// TwinCAT 3 PLC project PLC
// ProgramVersion: 3.1.4026.20
// CompilerDefines: VISU_USEPROPERTYINFO
// libraries:
//   SPT Base Types, * (Beckhoff Automation LLC)
//   SPT Components, * (Beckhoff Automation LLC)
//   SPT Diagnostic, * (Beckhoff Automation LLC)
//   SPT EtherCat, * (Beckhoff Automation LLC)
//   SPT Event Logger, * (Beckhoff Automation LLC)
//   SPT Motion Control, * (Beckhoff Automation LLC)
//   SPT Utilities, * (Beckhoff Automation LLC)
//   Tc2_MC2, * (Beckhoff Automation GmbH)
//   Tc2_MC2_Camming, * (Beckhoff Automation GmbH)
//   Tc2_Standard, * (Beckhoff Automation GmbH)
//   Tc2_System, * (Beckhoff Automation GmbH)
//   Tc2_Utilities, * (Beckhoff Automation GmbH)
//   Tc3_EventLogger, * (Beckhoff Automation GmbH)
//   Tc3_MC2_AdvancedHoming, * (Beckhoff Automation GmbH)
//   Tc3_McCollisionAvoidance, * (Beckhoff Automation GmbH)
//   Tc3_McCoordinatedMotion, * (Beckhoff Automation GmbH)
//   Tc3_PackML_V3, * (Beckhoff Automation GmbH)
// project tree:
//   / GlobalTextList.TcGTLO, PlcTask.TcTTO (not stored), VisualizationManager.TcVMO (not stored)
//   GVLs/ GVL.TcGVL (not stored)
//   POUs/BeltIndexer/ FB_DataSetFifo.TcPOU (not stored), FB_BeltIndexer.TcPOU
//   POUs/Camming/02 Cam Module Update Table/ CamModule_UpdateTable.TcPOU (not stored)
//   POUs/Camming/02 Cam Module Update Table/DUTs/ ST_EM_Cfg_UpdateTable.TcDUT, ST_EM_Cmd_UpdateTable.TcDUT, ST_EM_HMI_UpdateTable.TcDUT (not stored), ST_EM_Sts_UpdateTable.TcDUT
//   POUs/ Machine.TcPOU (not stored), MAIN.TcPOU (not stored)
//   POUs/RackAndPinion/ FB_RackAndPinion.TcPOU, FB_SwitchHoming.TcPOU, FB_TorqueHoming.TcPOU
//   POUs/Stitcher/ FB_Stitcher.TcPOU (not stored)
//   VISUs/ Visualization.TcVIS (not stored)

// ---- POUs/Camming/02 Cam Module Update Table/DUTs/ST_EM_Cfg_UpdateTable.TcDUT
TYPE ST_EM_Cfg_UpdateTable :
	STRUCT
		CamActivationMode : INT;
	END_STRUCT
END_TYPE

// ---- POUs/Camming/02 Cam Module Update Table/DUTs/ST_EM_Cmd_UpdateTable.TcDUT
TYPE ST_EM_Cmd_UpdateTable :
	STRUCT
		ChangeTable : BOOL;
		ChangeMode	: BOOL;
	END_STRUCT
END_TYPE

// ---- POUs/Camming/02 Cam Module Update Table/DUTs/ST_EM_Sts_UpdateTable.TcDUT
TYPE ST_EM_Sts_UpdateTable :
	STRUCT
		CurrentTable : UDINT;
	END_STRUCT
END_TYPE

// ---- POUs/RackAndPinion/FB_RackAndPinion.TcPOU
FUNCTION_BLOCK FB_RackAndPinion EXTENDS FB_PackML_BaseModule
VAR
	LeftAxis	: FB_Component_BasicAxis;
	RightAxis	: FB_Component_BasicAxis;

	TorqueHoming	: FB_TorqueHoming;
	SwitchHoming	: FB_SwitchHoming;

	// CA Group
	CAGroup			: AXES_GROUP_REF;
	GroupReadStatus	: MC_GroupReadStatus;
	GroupReset		: MC_GroupReset;
	GroupEnable		: MC_GroupEnable;
	GroupDisable	: MC_GroupDisable;
	AddToGroup		: ARRAY[0..1] OF MC_AddAxisToGroup;
	MoveAbsoluteCA	: ARRAY[0..1] OF MC_MoveAbsoluteCA;

	TON_Dwell	: TON;
END_VAR

//! @summary This method contains code which will execute when this PackML module is in the <b>Aborting</b> state
METHOD PROTECTED Aborting
VAR
	i				: UDINT;
	SubModulesReady : BOOL := TRUE;
END_VAR
CASE DescendantSequenceState OF
	0:
		NoStateTasksToComplete := FALSE;
		DescendantSequenceState := DescendantSequenceState + 10;

	10:
		IF LeftAxis.Disable() AND RightAxis.Disable() THEN
			StateTasksComplete 		:= TRUE;
			DescendantSequenceState := DescendantSequenceState + 10;
		END_IF

	//20:	

	20:
		StateTasksComplete := TRUE;
END_CASE

SUPER^.Aborting();
END_METHOD

//! @summary This method contains code which will execute when this PackML module is in the <b>Clearing</b> state
METHOD PROTECTED Clearing
VAR
	i				: UDINT;
	SubModulesReady : BOOL := TRUE;
END_VAR

VAR_INST

END_VAR

(*! <description> <b>Note:</b> The <i>Clear</i> command can also be thought of as a <i>fault reset</i> depite the ambiguity in the naming of the <i>Reset</i> state. 
<table> 
	<tr>
		<th> Previous State </th>
		<th> Transition In </th>
		<th> Transition Out </th>
		<th> Next State  </th> 
	</tr>
	<tr>
		<td> Aborted </td>
		<td> Clear Command </td> 
		<td> State Complete </td>
		<td> Stopped </td> 
	</tr>
</table>
This method is called as required by <c>StateControl()</c>
</description> 

*)
// CASE _CurrentMode OF
// 	E_PMLUnitMode.ePMLUnitMode_Production:
		CASE DescendantSequenceState OF
			0: //Init
				NoStateTasksToComplete := FALSE;

				//Reset Axes and  CA Group
				LeftAxis.Reset();
				RightAxis.Reset();
				GroupReset.Execute	:= TRUE;
				DescendantSequenceState := DescendantSequenceState + 10;

			10: // Done	
				GroupReset.Execute	:= FALSE;
				StateTasksComplete := TRUE;
		END_CASE

// END_CASE

SUPER^.Clearing();
END_METHOD

METHOD CyclicLogic
VAR_INPUT
END_VAR
SUPER^.CyclicLogic();

AddToGroup[0](Axis := LeftAxis.Axis, AxesGroup := CAGroup);
AddToGroup[1](Axis := RightAxis.Axis, AxesGroup := CAGroup);
GroupEnable(AxesGroup := CAGroup);
GroupDisable(AxesGroup := CAGroup);
GroupReadStatus.Enable		:= TRUE;
GroupReadStatus(AxesGroup	:= CAGroup);
GroupReset(AxesGroup	:= CAGroup);
MoveAbsoluteCA[0](Axis := LeftAxis.Axis);
MoveAbsoluteCA[1](Axis := RightAxis.Axis);
TON_Dwell();

TorqueHoming.CyclicLogic();
SwitchHoming.CyclicLogic();
END_METHOD

//! @summary This method contains code which will execute when this PackML module is in the <b>Execute</b> state
METHOD PROTECTED Execute
VAR
	i : UDINT;
END_VAR
(*CASE _CurrentMode OF
	E_PMLUnitMode.ePMLUnitMode_Production:


	E_PMLUnitMode.ePMLUnitMode_Manual:
		; //Insert logic for Manual Mode here
END_CASE	*)

CASE DescendantSequenceState OF
	0:
		FOR i := 0 TO 1 DO
			MoveAbsoluteCA[i].Execute		:= TRUE;
			MoveAbsoluteCA[i].Position		:= 50.0;
			MoveAbsoluteCA[i].Velocity		:= leftAxis.Velocity;
			MoveAbsoluteCA[i].Acceleration	:= LeftAxis.Acceleration;
			MoveAbsoluteCA[i].Deceleration	:= LeftAxis.Deceleration;
			MoveAbsoluteCA[i].Jerk			:= LeftAxis.Jerk;
			MoveAbsoluteCA[i].Gap			:= 68.0;
			MoveAbsoluteCA[i].Options.GapControlMode	:= MC_GAP_CONTROL_MODE.mcGapControlModeFast;
			MoveAbsoluteCA[i].BufferMode	:= mcAborting;
		END_FOR
		DescendantSequenceState				:= DescendantSequenceState + 10;

	10:	IF MoveAbsoluteCA[0].Done OR MoveAbsoluteCA[1].Done THEN
			MoveAbsoluteCA[0].Execute		:= FALSE;
			MoveAbsoluteCA[1].Execute		:= FALSE;
			TON_Dwell.IN	:= TRUE;
			TON_Dwell.PT	:= T#1S;
			DescendantSequenceState			:= DescendantSequenceState + 10;
		END_IF

	20: IF TON_Dwell.Q THEN
			ton_dwell.IN	:= FALSE;
			DescendantSequenceState			:= DescendantSequenceState + 10;
		END_IF

	30:
		FOR i := 0 TO 1 DO
			MoveAbsoluteCA[i].Execute		:= TRUE;
			MoveAbsoluteCA[i].Position		:= 450.0;
			MoveAbsoluteCA[i].Velocity		:= leftAxis.Velocity;
			MoveAbsoluteCA[i].Acceleration	:= LeftAxis.Acceleration;
			MoveAbsoluteCA[i].Deceleration	:= LeftAxis.Deceleration;
			MoveAbsoluteCA[i].Jerk			:= LeftAxis.Jerk;
			MoveAbsoluteCA[i].Gap			:= 68.0;
			MoveAbsoluteCA[i].Options.GapControlMode	:= MC_GAP_CONTROL_MODE.mcGapControlModeStandard;
			MoveAbsoluteCA[i].BufferMode	:= mcAborting;
		END_FOR
		DescendantSequenceState				:= DescendantSequenceState + 10;

	40:	IF MoveAbsoluteCA[0].Done OR MoveAbsoluteCA[1].Done THEN
			MoveAbsoluteCA[0].Execute		:= FALSE;
			MoveAbsoluteCA[1].Execute		:= FALSE;
			TON_Dwell.IN	:= TRUE;
			TON_Dwell.PT	:= T#1S;
			DescendantSequenceState			:= DescendantSequenceState + 10;

		END_IF

	50: IF TON_Dwell.Q THEN
			ton_dwell.IN	:= FALSE;
			DescendantSequenceState			:= 0;
		END_IF

END_CASE
END_METHOD

(* Basic module initialization logic*)
METHOD PROTECTED Initialize : BOOL
Initialize := FALSE;
CASE DescendantSequenceState OF
	0:
		RegisterComponent(Component := LeftAxis);
		RegisterComponent(Component := RightAxis);
		DescendantSequenceState := DescendantSequenceState + 10;

	10:
		IF SUPER^.Initialize() THEN
			DescendantSequenceState := DescendantSequenceState + 10;
		END_IF

	20:
		Initialize := TRUE;
END_CASE
END_METHOD

METHOD PROTECTED Resetting
VAR_INST
	i			 : UDINT;
END_VAR
// CASE _CurrentMode OF
// 	E_PMLUnitMode.ePMLUnitMode_Production:
		CASE DescendantSequenceState OF
			0: //Init
				i					   := 1;
				NoStateTasksToComplete := FALSE;
				DescendantSequenceState := DescendantSequenceState + 10;

			10: //Enable Axes
				IF LeftAxis.Enable() AND RightAxis.Enable() THEN
					DescendantSequenceState := DescendantSequenceState + 10;
				END_IF

			// Add logic to home left axis to switch and right axis to hard stop
			20: // Home Right Axis
				TorqueHoming.Axis	:= RightAxis;
				SwitchHoming.Axis	:= LeftAxis;
				IF TorqueHoming.Execute() AND SwitchHoming.Execute() THEN
					DescendantSequenceState := DescendantSequenceState + 20;
				END_IF

			30:	// Home Left Axis
				SwitchHoming.Axis	:= LeftAxis;
				IF SwitchHoming.Execute() THEN
					DescendantSequenceState := DescendantSequenceState + 10;
				END_IF

			40: //Add Movers to Group			
				AddToGroup[0].Execute		:= AddToGroup[1].Execute		:= TRUE;
				AddToGroup[0].IdentInGroup	:= UDINT_TO_IDENTINGROUP(1);
				AddToGroup[1].IdentInGroup	:= UDINT_TO_IDENTINGROUP(2);
				IF AddToGroup[0].Done AND AddToGroup[1].Done THEN	
					AddToGroup[0].Execute	:= AddToGroup[1].Execute	:= FALSE;
					DescendantSequenceState := DescendantSequenceState + 10;
				END_IF

			50: //Enable CA Group
				GroupEnable.Execute	:= TRUE;
				IF GroupEnable.Done THEN
					DescendantSequenceState := DescendantSequenceState + 10;
				END_IF

			60: //Clearing complete
				StateTasksComplete := TRUE;

		END_CASE
// END_CASE

SUPER^.Resetting();
END_METHOD

METHOD PROTECTED Starting
VAR_INST
	i		  : UDINT;
END_VAR
//CASE _CurrentMode OF
//	E_PMLUnitMode.ePMLUnitMode_Production:
		CASE DescendantSequenceState OF
			0:
				NoStateTasksToComplete	:= FALSE;
				DescendantSequenceState := 10;
				i						:= 1;

			10: //Set Axis Parameters
				LeftAxis.Velocity		:= 250;		RightAxis.Velocity		:= 250;
				LeftAxis.Acceleration	:= 1000;	RightAxis.Acceleration	:= 1000;
				LeftAxis.Deceleration	:= 1000;	RightAxis.Deceleration	:= 1000;
				LeftAxis.Jerk			:= 10000;	RightAxis.Jerk			:= 10000;
				DescendantSequenceState := DescendantSequenceState + 10;
				StateTasksComplete 		:= TRUE;

			20: //Cleanup mover queues
				DescendantSequenceState := DescendantSequenceState + 10;

		END_CASE

	//E_PMLUnitMode.ePMLUnitMode_Manual:
//END_CASE

SUPER^.Starting();
END_METHOD

END_FUNCTION_BLOCK

// ---- POUs/RackAndPinion/FB_TorqueHoming.TcPOU
FUNCTION_BLOCK FB_TorqueHoming IMPLEMENTS I_MotionSequence
VAR_INPUT
	HomingParameter	: MC_HomingParameter;
END_VAR
VAR_OUTPUT
	State	: UINT;
END_VAR
VAR
	validaxisref	: BOOL := FALSE;
	_Axis			: SPT_Motion_Control.I_BasicAxis;
	StepBlockHoming	: MC_StepBlock;
	FinishHoming	: MC_FinishHoming;
END_VAR

{warning 'Add property implementation'}
PROPERTY Axis : SPT_Motion_Control.I_BasicAxis
GET
Axis	:= _Axis;
END_GET
SET
_Axis	:= Axis;
validaxisref	:= TRUE;
END_SET
END_PROPERTY

{warning 'Add property implementation'}
PROPERTY Busy : BOOL
GET
END_GET
END_PROPERTY

{warning 'Add method implementation '}
METHOD CyclicLogic
IF validaxisref THEN
	StepBlockHoming(Axis := _Axis.Axis, Parameter := HomingParameter);
	FinishHoming(Axis := _Axis.Axis, Parameter := HomingParameter);
END_IF

IF NOT StepBlockHoming.Execute	THEN
	State	:= 0;
END_IF
StepBlockHoming.Execute	:= FALSE;
FinishHoming.Execute	:= FALSE;
END_METHOD

{warning 'Add property implementation'}
PROPERTY Error : BOOL
GET
END_GET
END_PROPERTY

{warning 'Add property implementation'}
PROPERTY ErrorID : UDINT
GET
END_GET
END_PROPERTY

{warning 'Add method implementation '}
METHOD Execute : BOOL
StepBlockHoming.Execute					:= TRUE;
StepBlockHoming.SetPosition				:= 472;
StepBlockHoming.Direction				:= mcPositiveDirection;
StepBlockHoming.Velocity				:= 50;
StepBlockHoming.Acceleration			:= 1000;
StepBlockHoming.Deceleration			:= 1000;
StepBlockHoming.Jerk					:= 10000;
StepBlockHoming.DetectionVelocityLimit	:= 1;
StepBlockHoming.DetectionVelocityTime	:= T#100MS;
StepBlockHoming.TimeLimit				:= T#10S;
StepBlockHoming.DistanceLimit			:= 500;
StepBlockHoming.TorqueLimit				:= 50;
StepBlockHoming.TorqueTolerance			:= 5;

FinishHoming.Execute		:= StepBlockHoming.Done;
FinishHoming.Distance		:= -0.5;
FinishHoming.Velocity		:= 100;
FinishHoming.Acceleration	:= 1000;
FinishHoming.Deceleration	:= 1000;
FinishHoming.Jerk			:= 1000;

// return true when done
Execute	:= StepBlockHoming.Done AND FinishHoming.Done;
END_METHOD

{warning 'Add property implementation'}
PROPERTY InitComplete : BOOL
GET
END_GET
END_PROPERTY

END_FUNCTION_BLOCK

// ---- POUs/RackAndPinion/FB_SwitchHoming.TcPOU
FUNCTION_BLOCK FB_SwitchHoming IMPLEMENTS I_MotionSequence
VAR_INPUT
	HomingParameter	: MC_HomingParameter;
END_VAR
VAR_OUTPUT
	State	: UINT;
END_VAR
VAR
	diHomeSwitch	AT %I* : BOOL;
	doHomeSwitch	AT %Q* : BOOL := TRUE;
	validaxisref	: BOOL := FALSE;
	_Axis			: SPT_Motion_Control.I_BasicAxis;
	Home			: MC_Home;
END_VAR

{warning 'Add property implementation'}
PROPERTY Axis : SPT_Motion_Control.I_BasicAxis
GET
Axis	:= _Axis;
END_GET
SET
_Axis	:= Axis;
validaxisref	:= TRUE;
END_SET
END_PROPERTY

{warning 'Add property implementation'}
PROPERTY Busy : BOOL
GET
END_GET
END_PROPERTY

{warning 'Add method implementation '}
METHOD CyclicLogic
IF validaxisref THEN
	Home.bCalibrationCam	:= diHomeSwitch;
	Home(Axis := _Axis.Axis);

END_IF

IF NOT Home.Execute	THEN
	State	:= 0;
END_IF
Home.Execute	:= FALSE;
END_METHOD

{warning 'Add property implementation'}
PROPERTY Error : BOOL
GET
END_GET
END_PROPERTY

{warning 'Add property implementation'}
PROPERTY ErrorID : UDINT
GET
END_GET
END_PROPERTY

{warning 'Add method implementation '}
METHOD Execute : BOOL
Home.Execute					:= TRUE;
Home.Position					:= 39;
Home.HomingMode					:= MC_DefaultHoming;
Home.Options.SearchVelocity		:= 50;
Home.Options.SearchDirection	:= MC_Negative_Direction;

// return true when done
Execute	:= Home.Done;
END_METHOD

{warning 'Add property implementation'}
PROPERTY InitComplete : BOOL
GET
END_GET
END_PROPERTY

END_FUNCTION_BLOCK

// ---- POUs/BeltIndexer/FB_BeltIndexer.TcPOU
FUNCTION_BLOCK FB_BeltIndexer EXTENDS FB_PackML_BaseModule
VAR
	BeltAxis	: FB_Component_BasicAxis;

	TouchProbe			: MC_TouchProbe;
	TouchProbeConfig	: TRIGGER_REF;
	fbFifo 				: FB_DataSetFifo := ( bOverwrite := TRUE );
	arrBuffer 			: ARRAY[0..MAX_BUFFER_SIZE] OF BYTE; (* Buffer memory used by FB_MemRingBuffer function block *)

	NewRecordedPosition	: LREAL;
	OldRecordedPosition	: LREAL;

	TON_Dwell	: TON;
END_VAR

//! @summary This method contains code which will execute when this PackML module is in the <b>Aborting</b> state
METHOD PROTECTED Aborting
VAR
	i				: UDINT;
	SubModulesReady : BOOL := TRUE;
END_VAR
CASE DescendantSequenceState OF
	0:
		NoStateTasksToComplete := FALSE;
		DescendantSequenceState := DescendantSequenceState + 10;

	10:
		IF BeltAxis.Disable() THEN
			TouchProbe.Execute		:= FALSE;
			NewRecordedPosition		:= 0;
			OldRecordedPosition		:= 0;
			StateTasksComplete 		:= TRUE;
			DescendantSequenceState := DescendantSequenceState + 10;
		END_IF

	//20:	

	20:
		StateTasksComplete := TRUE;
END_CASE

SUPER^.Aborting();
END_METHOD

//! @summary This method contains code which will execute when this PackML module is in the <b>Clearing</b> state
METHOD PROTECTED Clearing
VAR
	i				: UDINT;
	SubModulesReady : BOOL := TRUE;
END_VAR

VAR_INST

END_VAR

(*! <description> <b>Note:</b> The <i>Clear</i> command can also be thought of as a <i>fault reset</i> depite the ambiguity in the naming of the <i>Reset</i> state. 
<table> 
	<tr>
		<th> Previous State </th>
		<th> Transition In </th>
		<th> Transition Out </th>
		<th> Next State  </th> 
	</tr>
	<tr>
		<td> Aborted </td>
		<td> Clear Command </td> 
		<td> State Complete </td>
		<td> Stopped </td> 
	</tr>
</table>
This method is called as required by <c>StateControl()</c>
</description> 

*)
// CASE _CurrentMode OF
// 	E_PMLUnitMode.ePMLUnitMode_Production:
		CASE DescendantSequenceState OF
			0: //Init
				NoStateTasksToComplete := FALSE;

				//Reset Axes and  CA Group
				BeltAxis.Reset();
				DescendantSequenceState := DescendantSequenceState + 10;

			10: // Done	
				StateTasksComplete := TRUE;
		END_CASE

// END_CASE

SUPER^.Clearing();
END_METHOD

METHOD CyclicLogic
VAR_INPUT
END_VAR
SUPER^.CyclicLogic();

TouchProbe(Axis := BeltAxis.Axis, TriggerInput := TouchProbeConfig);
fbFifo();
TON_Dwell();
END_METHOD

//! @summary This method contains code which will execute when this PackML module is in the <b>Execute</b> state
METHOD PROTECTED Execute
VAR
	i : UDINT;
END_VAR
(*CASE _CurrentMode OF
	E_PMLUnitMode.ePMLUnitMode_Production:


	E_PMLUnitMode.ePMLUnitMode_Manual:
		; //Insert logic for Manual Mode here
END_CASE	*)

CASE DescendantSequenceState OF
	0:	// Start Moving
		BeltAxis.MoveVelocity(250, TRUE);
		TouchProbe.Execute		:= TRUE;
		DescendantSequenceState	:= DescendantSequenceState + 10;

	10: // Start buffering positions and moving to them
		IF fbFifo.nCount > 0 THEN
			fbFifo.A_Get(out => OldRecordedPosition);
			BeltAxis.MoveAbsolute(OldRecordedPosition + 440.0, TRUE);
			DescendantSequenceState	:= DescendantSequenceState + 10;
		END_IF
		
	20: // Look for trigger
		IF ton_dwell.Q THEN
			TON_Dwell.IN			:= FALSE;
			fbFifo.A_Remove();
			IF fbFifo.nCount > 0 THEN
				DescendantSequenceState	:= 10;
			ELSE
				DescendantSequenceState	:= 0;
			END_IF
		ELSIF BeltAxis.InPosition AND (ABS(BeltAxis.SetPosition - (OldRecordedPosition + 440)) < 1) THEN
			Ton_Dwell.IN	:= TRUE;
		END_IF

END_CASE

IF TouchProbe.Done THEN
	NewRecordedPosition	:= TouchProbe.RecordedData.AbsolutePosition;
	fbFifo.A_Add(In := NewRecordedPosition);
END_IF
END_METHOD

(* Basic module initialization logic*)
METHOD PROTECTED Initialize : BOOL
Initialize := FALSE;
CASE DescendantSequenceState OF
	0:
		RegisterComponent(Component := BeltAxis);
		DescendantSequenceState := DescendantSequenceState + 10;

	10: // Touch Probe Configuration
		TouchProbeConfig.SignalSource	:= SignalSource_DriveDefined;
		TouchProbeconfig.Mode			:= TOUCHPROBEMODE_CONTINOUS;
		TON_Dwell.PT					:= T#500ms;
		DescendantSequenceState 		:= DescendantSequenceState + 10;

	20:
		IF SUPER^.Initialize() THEN
			DescendantSequenceState := DescendantSequenceState + 10;
		END_IF

	30:
		Initialize := TRUE;
END_CASE
END_METHOD

METHOD PROTECTED Resetting
VAR_INST
	i			 : UDINT;
END_VAR
// CASE _CurrentMode OF
// 	E_PMLUnitMode.ePMLUnitMode_Production:
		CASE DescendantSequenceState OF
			0: //Init
				i					   := 1;
				NoStateTasksToComplete := FALSE;
				DescendantSequenceState := DescendantSequenceState + 10;

			10: //Enable Axes
				IF BeltAxis.Enable() THEN
					DescendantSequenceState := DescendantSequenceState + 10;
				END_IF

			20:	// Home Axis
				IF BeltAxis.Home() THEN
					DescendantSequenceState := DescendantSequenceState + 10;
				END_IF
	
			30: // Clear Buffer
				fbFifo.A_Reset();
				DescendantSequenceState := DescendantSequenceState + 10;

			40: //Clearing complete
				StateTasksComplete := TRUE;

		END_CASE
// END_CASE

SUPER^.Resetting();
END_METHOD

METHOD PROTECTED Starting
VAR_INST
	i		  : UDINT;
END_VAR
//CASE _CurrentMode OF
//	E_PMLUnitMode.ePMLUnitMode_Production:
		CASE DescendantSequenceState OF
			0:
				NoStateTasksToComplete	:= FALSE;
				DescendantSequenceState := 10;
				i						:= 1;

			10: //Set Axis Parameters
				BeltAxis.Velocity		:= 500;
				BeltAxis.Acceleration	:= 1000;
				BeltAxis.Deceleration	:= 1000;
				BeltAxis.Jerk			:= 10000;
				DescendantSequenceState := DescendantSequenceState + 10;

			20: // Start Touchprobe and clear buffer
				TouchProbe.WindowOnly		:= FALSE;
				TouchProbeConfig.EncoderID	:= 4;
				DescendantSequenceState 	:= DescendantSequenceState + 10;
				
			30: // Finsihed
				StateTasksComplete 		:= TRUE;

		END_CASE

	//E_PMLUnitMode.ePMLUnitMode_Manual:
//END_CASE

SUPER^.Starting();
END_METHOD

END_FUNCTION_BLOCK
